      A(    ;
      O     I      0.2;
      O     M   1802.0;
      O     M    201.5;
      )     ;
      AN    M    201.7;
      A     M    201.6;
      A     M   1800.0;
      AN    M   1700.0;
      =     L      0.0;
      A     L      0.0;
      BLD   102;
      =     M    201.5;
      A     L      0.0;
      A     I      0.0;
      AN    I      0.1;
      =     M    201.4;
      A     L      0.0;
      AN    I      0.0;
      AN    I      0.1;
      =     M    202.0;
      A     L      0.0;
      AN    I      0.0;
      A     I      0.1;
      =     M    201.3;
NETWORK
TITLE =AUTO START

      A(    ;
      O     I      0.5;
      O     M   1802.1;
      O     M    201.2;
      )     ;
      A     M    201.4;
      A     I     68.1;
      A     I     69.0;
      AN    M    200.7;
      =     M    201.2;
NETWORK
TITLE =

      AN    M    201.7;
      AN    M    202.5;
      AN    M    601.1;
      AN    M    200.6;
      AN    M    820.0;
      NOT   ;
      =     M    200.7;
NETWORK
TITLE =AIR ERROR

      ON    I     31.2;
      O     ;
      A     M    201.7;
      AN    M    201.1;
      =     M    201.7;
NETWORK
TITLE =
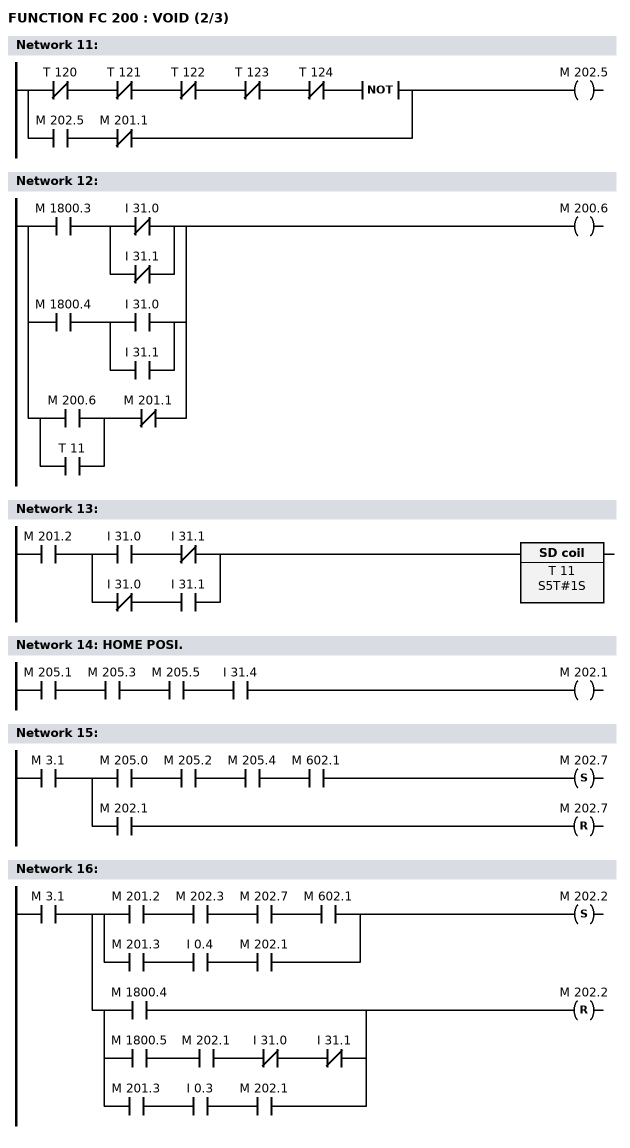

      AN    T    120;
      AN    T    121;
      AN    T    122;
      AN    T    123;
      AN    T    124;
      NOT   ;
      O     ;
      A     M    202.5;
      AN    M    201.1;
      =     M    202.5;
NETWORK
TITLE =

      A     M   1800.3;
      A(    ;
      ON    I     31.0;
      ON    I     31.1;
      )     ;
      O     ;
      A     M   1800.4;
      A(    ;
      O     I     31.0;
      O     I     31.1;
      )     ;
      O     ;
      A(    ;
      O     M    200.6;
      O     T     11;
      )     ;
      AN    M    201.1;
      =     M    200.6;
NETWORK
TITLE =

      A     M    201.2;
      A(    ;
      A     I     31.0;
      AN    I     31.1;
      O     ;
      AN    I     31.0;
      A     I     31.1;
      )     ;
      L     S5T#1S;
      SD    T     11;
NETWORK
TITLE =HOME POSI.

      A     M    205.1;
      A     M    205.3;
      A     M    205.5;
      A     I     31.4;
      =     M    202.1;
NETWORK
TITLE =

      A     M      3.1;
      =     L      0.0;
      A     L      0.0;
      A     M    205.0;
      A     M    205.2;
      A     M    205.4;
      A     M    602.1;
      S     M    202.7;
      A     L      0.0;
      A     M    202.1;
      R     M    202.7;
NETWORK
TITLE =

      A     M      3.1;
      =     L      0.0;
      A     L      0.0;
      A(    ;
      A     M    201.2;
      A     M    202.3;
      A     M    202.7;
      A     M    602.1;
      O     ;
      A     M    201.3;
      A     I      0.4;
      A     M    202.1;
      )     ;
      S     M    202.2;
      A     L      0.0;
      A(    ;
      O     M   1800.4;
      O     ;
      A     M   1800.5;
      A     M    202.1;
      AN    I     31.0;
      AN    I     31.1;
      O     ;
      A     M    201.3;
      A     I      0.3;
      A     M    202.1;
      )     ;
      R     M    202.2;
NETWORK
TITLE =
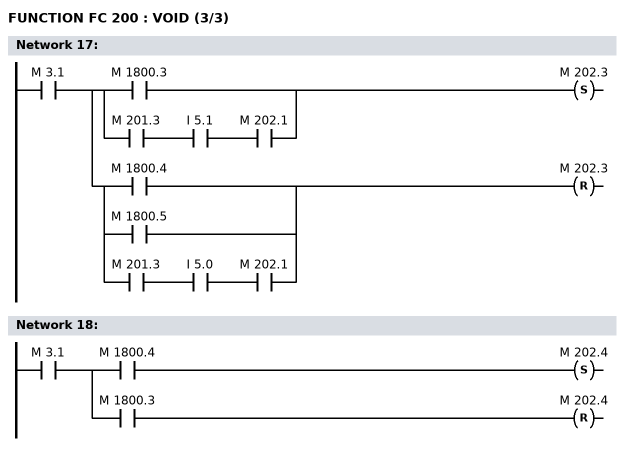

      A     M      3.1;
      =     L      0.0;
      A     L      0.0;
      A(    ;
      O     M   1800.3;
      O     ;
      A     M    201.3;
      A     I      5.1;
      A     M    202.1;
      )     ;
      S     M    202.3;
      A     L      0.0;
      A(    ;
      O     M   1800.4;
      O     M   1800.5;
      O     ;
      A     M    201.3;
      A     I      5.0;
      A     M    202.1;
      )     ;
      R     M    202.3;
NETWORK
TITLE =

      A     M      3.1;
      =     L      0.0;
      A     L      0.0;
      A     M   1800.4;
      S     M    202.4;
      A     L      0.0;
      A     M   1800.3;
      R     M    202.4;
NETWORK
TITLE =

      AN    OV;
      =     L      0.0;
      A     L      0.0;
      A(    ;
      O     M   1800.4;
      O     M   1801.0;
      )     ;
      S     M    207.0;
      A     L      0.0;
      A     T     70;
      R     M    207.0;
NETWORK
TITLE =CAM1 UP

      A     M    201.3;
      =     L      0.0;
      A     L      0.0;
      AN    I      3.5;
      =     L      0.1;
      A     L      0.1;
      AN    I      3.4;
      =     L      0.2;
      A     L      0.2;
      AN    I      3.3;
      A     I      3.2;
      =     M    203.0;
      A     L      0.2;
      A     I      3.3;
      AN    I      3.2;
      =     M    203.1;
      A     L      0.2;
      A     I      3.3;
      A     I      3.2;
      =     M    203.2;
      A     L      0.1;
      A     I      3.4;
      =     L      0.2;
      A     L      0.2;
      AN    I      3.3;
      =     L      0.3;
      A     L      0.3;
      AN    I      3.2;
      =     M    203.3;
      A     L      0.3;
      A     I      3.2;
      =     M    203.4;
      A     L      0.2;
      A     I      3.3;
      =     L      0.3;
      A     L      0.3;
      AN    I      3.2;
      =     M    203.5;
      A     L      0.3;
      A     I      3.2;
      =     M    203.6;
      A     L      0.0;
      A     I      3.4;
      AN    I      3.4;
      =     L      0.1;
      A     L      0.1;
      AN    I      3.3;
      =     L      0.2;
      A     L      0.2;
      AN    I      3.2;
      =     M    203.7;
      A     L      0.2;
      A     I      3.2;
      =     M    204.0;
      A     L      0.1;
      A     I      3.3;
      =     L      0.2;
      A     L      0.2;
      AN    I      3.2;
      =     M    204.1;
      A     L      0.2;
      A     I      3.2;
      =     M    204.2;
NETWORK
TITLE =핀/클램프 전_후진단
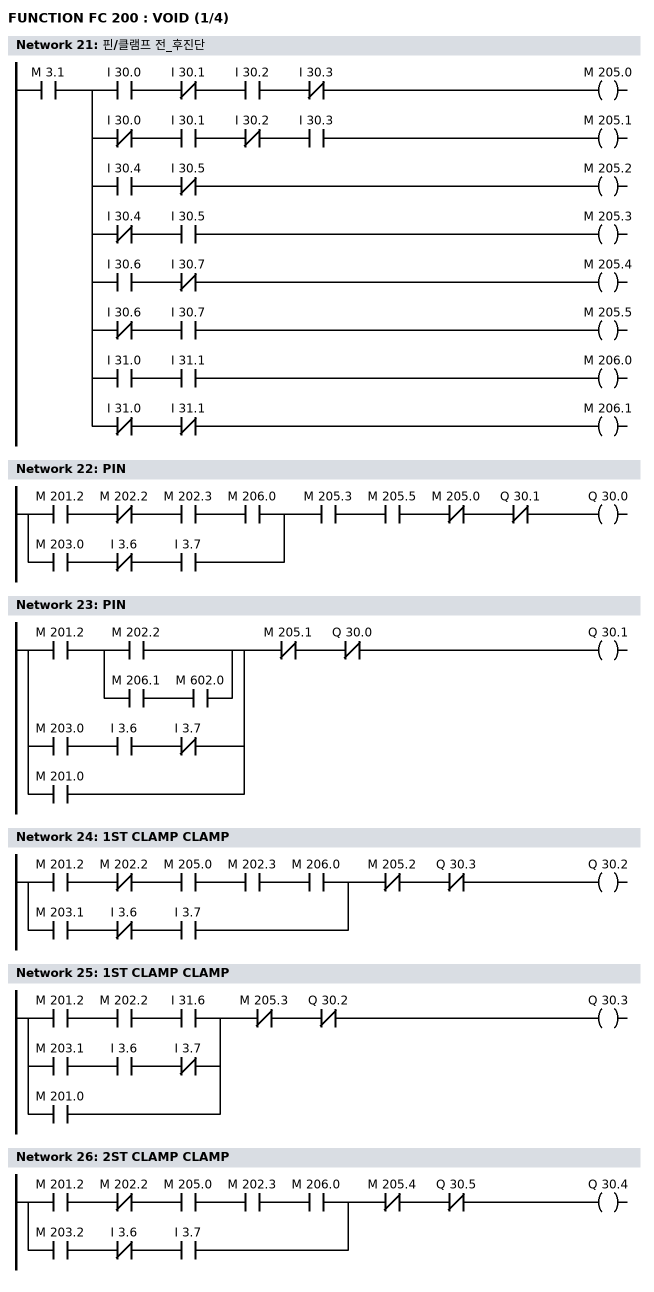

      A     M      3.1;
      =     L      0.0;
      A     L      0.0;
      A     I     30.0;
      AN    I     30.1;
      A     I     30.2;
      AN    I     30.3;
      =     M    205.0;
      A     L      0.0;
      AN    I     30.0;
      A     I     30.1;
      AN    I     30.2;
      A     I     30.3;
      =     M    205.1;
      A     L      0.0;
      A     I     30.4;
      AN    I     30.5;
      =     M    205.2;
      A     L      0.0;
      AN    I     30.4;
      A     I     30.5;
      =     M    205.3;
      A     L      0.0;
      A     I     30.6;
      AN    I     30.7;
      =     M    205.4;
      A     L      0.0;
      AN    I     30.6;
      A     I     30.7;
      =     M    205.5;
      A     L      0.0;
      A     I     31.0;
      A     I     31.1;
      =     M    206.0;
      A     L      0.0;
      AN    I     31.0;
      AN    I     31.1;
      =     M    206.1;
NETWORK
TITLE =PIN

      A(    ;
      A     M    201.2;
      AN    M    202.2;
      A     M    202.3;
      A     M    206.0;
      O     ;
      A     M    203.0;
      AN    I      3.6;
      A     I      3.7;
      )     ;
      A     M    205.3;
      A     M    205.5;
      AN    M    205.0;
      AN    Q     30.1;
      =     Q     30.0;
NETWORK
TITLE =PIN

      A(    ;
      A     M    201.2;
      A(    ;
      O     M    202.2;
      O     ;
      A     M    206.1;
      A     M    602.0;
      )     ;
      O     ;
      A     M    203.0;
      A     I      3.6;
      AN    I      3.7;
      O     M    201.0;
      )     ;
      AN    M    205.1;
      AN    Q     30.0;
      =     Q     30.1;
NETWORK
TITLE =1ST CLAMP CLAMP

      A(    ;
      A     M    201.2;
      AN    M    202.2;
      A     M    205.0;
      A     M    202.3;
      A     M    206.0;
      O     ;
      A     M    203.1;
      AN    I      3.6;
      A     I      3.7;
      )     ;
      AN    M    205.2;
      AN    Q     30.3;
      =     Q     30.2;
NETWORK
TITLE =1ST CLAMP CLAMP

      A(    ;
      A     M    201.2;
      A     M    202.2;
      A     I     31.6;
      O     ;
      A     M    203.1;
      A     I      3.6;
      AN    I      3.7;
      O     M    201.0;
      )     ;
      AN    M    205.3;
      AN    Q     30.2;
      =     Q     30.3;
NETWORK
TITLE =2ST CLAMP CLAMP

      A(    ;
      A     M    201.2;
      AN    M    202.2;
      A     M    205.0;
      A     M    202.3;
      A     M    206.0;
      O     ;
      A     M    203.2;
      AN    I      3.6;
      A     I      3.7;
      )     ;
      AN    M    205.4;
      AN    Q     30.5;
      =     Q     30.4;
NETWORK
TITLE =2ST CLAMP CLAMP
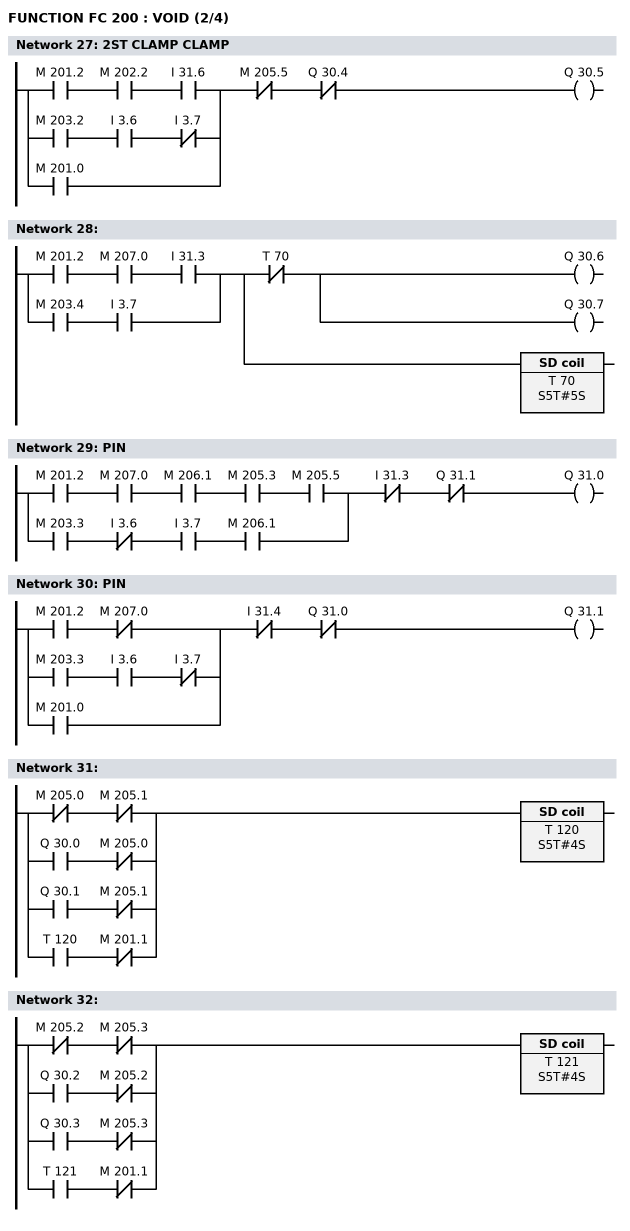

      A(    ;
      A     M    201.2;
      A     M    202.2;
      A     I     31.6;
      O     ;
      A     M    203.2;
      A     I      3.6;
      AN    I      3.7;
      O     M    201.0;
      )     ;
      AN    M    205.5;
      AN    Q     30.4;
      =     Q     30.5;
NETWORK
TITLE =

      A     M    201.2;
      A     M    207.0;
      A     I     31.3;
      O     ;
      A     M    203.4;
      A     I      3.7;
      =     L      0.0;
      A     L      0.0;
      AN    T     70;
      =     Q     30.6;
      =     Q     30.7;
      A     L      0.0;
      BLD   102;
      L     S5T#5S;
      SD    T     70;
NETWORK
TITLE =PIN

      A(    ;
      A     M    201.2;
      A     M    207.0;
      A     M    206.1;
      A     M    205.3;
      A     M    205.5;
      O     ;
      A     M    203.3;
      AN    I      3.6;
      A     I      3.7;
      A     M    206.1;
      )     ;
      AN    I     31.3;
      AN    Q     31.1;
      =     Q     31.0;
NETWORK
TITLE =PIN

      A(    ;
      A     M    201.2;
      AN    M    207.0;
      O     ;
      A     M    203.3;
      A     I      3.6;
      AN    I      3.7;
      O     M    201.0;
      )     ;
      AN    I     31.4;
      AN    Q     31.0;
      =     Q     31.1;
NETWORK
TITLE =

      AN    M    205.0;
      AN    M    205.1;
      O     ;
      A     Q     30.0;
      AN    M    205.0;
      O     ;
      A     Q     30.1;
      AN    M    205.1;
      O     ;
      A     T    120;
      AN    M    201.1;
      L     S5T#4S;
      SD    T    120;
NETWORK
TITLE =

      AN    M    205.2;
      AN    M    205.3;
      O     ;
      A     Q     30.2;
      AN    M    205.2;
      O     ;
      A     Q     30.3;
      AN    M    205.3;
      O     ;
      A     T    121;
      AN    M    201.1;
      L     S5T#4S;
      SD    T    121;
NETWORK
TITLE =
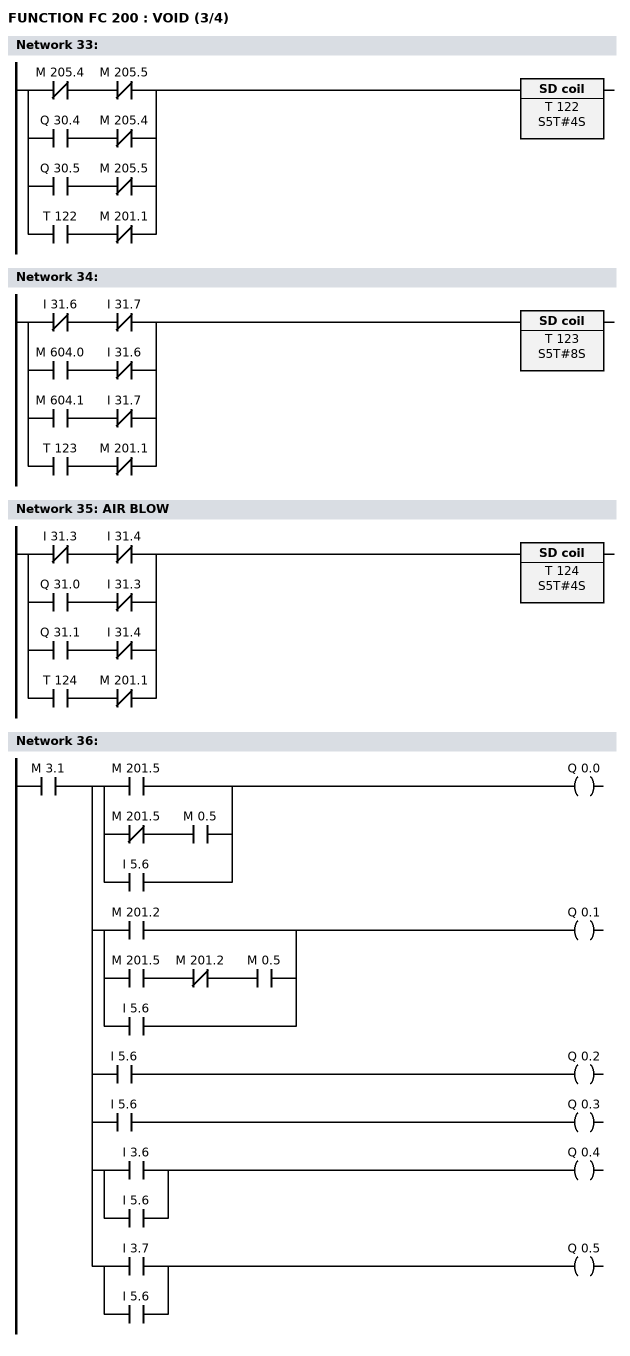

      AN    M    205.4;
      AN    M    205.5;
      O     ;
      A     Q     30.4;
      AN    M    205.4;
      O     ;
      A     Q     30.5;
      AN    M    205.5;
      O     ;
      A     T    122;
      AN    M    201.1;
      L     S5T#4S;
      SD    T    122;
NETWORK
TITLE =

      AN    I     31.6;
      AN    I     31.7;
      O     ;
      A     M    604.0;
      AN    I     31.6;
      O     ;
      A     M    604.1;
      AN    I     31.7;
      O     ;
      A     T    123;
      AN    M    201.1;
      L     S5T#8S;
      SD    T    123;
NETWORK
TITLE =AIR BLOW

      AN    I     31.3;
      AN    I     31.4;
      O     ;
      A     Q     31.0;
      AN    I     31.3;
      O     ;
      A     Q     31.1;
      AN    I     31.4;
      O     ;
      A     T    124;
      AN    M    201.1;
      L     S5T#4S;
      SD    T    124;
NETWORK
TITLE =

      A     M      3.1;
      =     L      0.0;
      A     L      0.0;
      A(    ;
      O     M    201.5;
      O     ;
      AN    M    201.5;
      A     M      0.5;
      O     I      5.6;
      )     ;
      =     Q      0.0;
      A     L      0.0;
      A(    ;
      O     M    201.2;
      O     ;
      A     M    201.5;
      AN    M    201.2;
      A     M      0.5;
      O     I      5.6;
      )     ;
      =     Q      0.1;
      A     L      0.0;
      A     I      5.6;
      =     Q      0.2;
      A     L      0.0;
      A     I      5.6;
      =     Q      0.3;
      A     L      0.0;
      A(    ;
      O     I      3.6;
      O     I      5.6;
      )     ;
      =     Q      0.4;
      A     L      0.0;
      A(    ;
      O     I      3.7;
      O     I      5.6;
      )     ;
      =     Q      0.5;
NETWORK
TITLE =메인제어반1 에어이상 램프
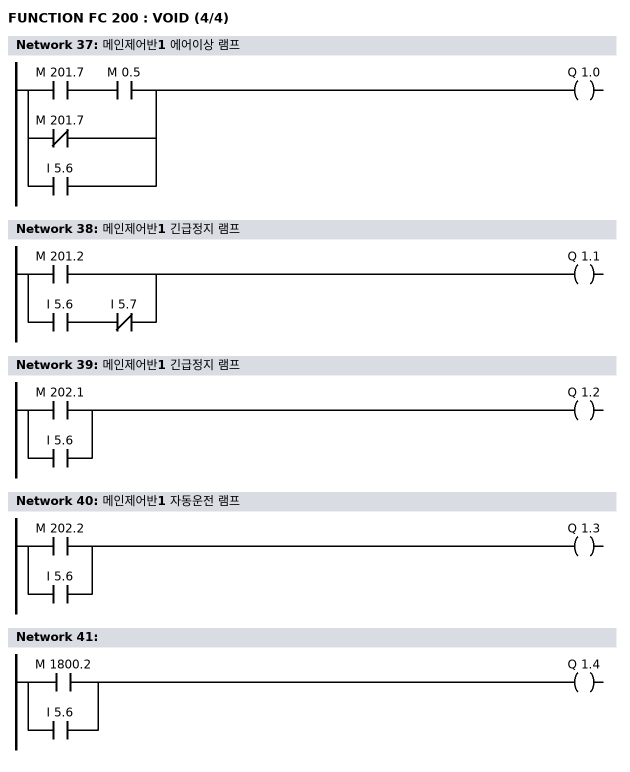

      A     M    201.7;
      A     M      0.5;
      ON    M    201.7;
      O     I      5.6;
      =     Q      1.0;
NETWORK
TITLE =메인제어반1 긴급정지 램프

      O     M    201.2;
      O     ;
      A     I      5.6;
      AN    I      5.7;
      =     Q      1.1;
NETWORK
TITLE =메인제어반1 긴급정지 램프

      O     M    202.1;
      O     I      5.6;
      =     Q      1.2;
NETWORK
TITLE =메인제어반1 자동운전 램프

      O     M    202.2;
      O     I      5.6;
      =     Q      1.3;
NETWORK
TITLE =

      O     M   1800.2;
      O     I      5.6;
      =     Q      1.4;
NETWORK
TITLE =

      A     DB486.DBX   21.1;
      A     OV;
      O     I      5.6;
      =     Q      1.5;
NETWORK
TITLE =
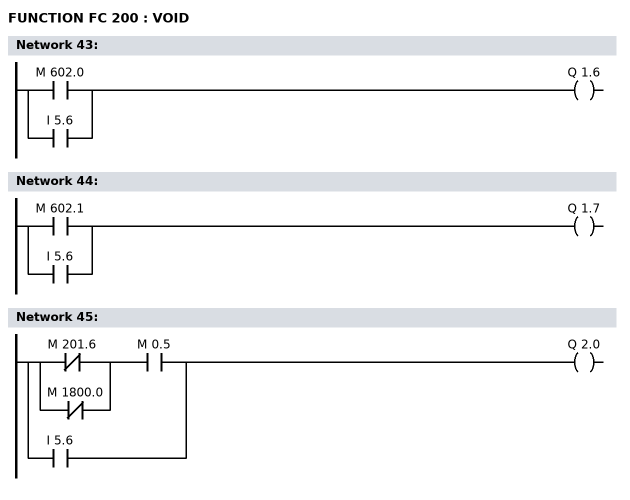

      O     M    602.0;
      O     I      5.6;
      =     Q      1.6;
NETWORK
TITLE =

      O     M    602.1;
      O     I      5.6;
      =     Q      1.7;
NETWORK
TITLE =

      A(    ;
      ON    M    201.6;
      ON    M   1800.0;
      )     ;
      A     M      0.5;
      O     I      5.6;
      =     Q      2.0;
NETWORK
TITLE =

      A     M    202.5;
      A     OV;
      O     I      5.6;
      =     Q      2.1;
NETWORK
TITLE =
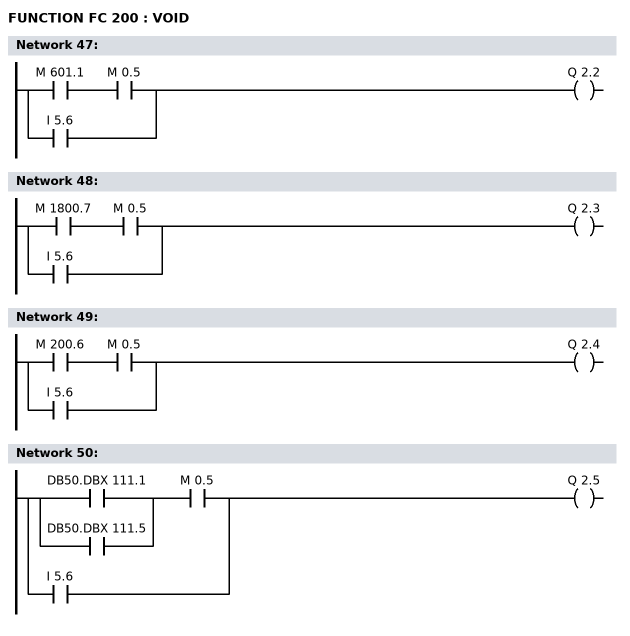

      A     M    601.1;
      A     M      0.5;
      O     I      5.6;
      =     Q      2.2;
NETWORK
TITLE =

      A     M   1800.7;
      A     M      0.5;
      O     I      5.6;
      =     Q      2.3;
NETWORK
TITLE =

      A     M    200.6;
      A     M      0.5;
      O     I      5.6;
      =     Q      2.4;
NETWORK
TITLE =

      A(    ;
      O     DB50.DBX  111.1;
      O     DB50.DBX  111.5;
      )     ;
      A     M      0.5;
      O     I      5.6;
      =     Q      2.5;
NETWORK
TITLE =

      A     OV;
      A     M      0.5;
      O     I      5.6;
      =     Q      2.6;
NETWORK
TITLE =

      A     OV;
      A     M      0.5;
      O     I      5.6;
      =     Q      2.7;
NETWORK
TITLE =부저울림
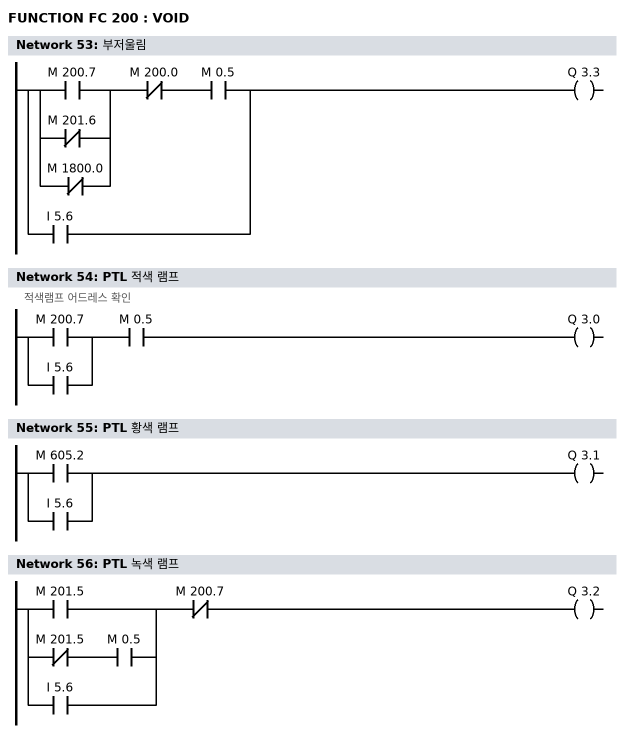

      A(    ;
      O     M    200.7;
      ON    M    201.6;
      ON    M   1800.0;
      )     ;
      AN    M    200.0;
      A     M      0.5;
      O     I      5.6;
      =     Q      3.3;
NETWORK
TITLE =PTL 적색 램프
//적색램프 어드레스 확인
      A(    ;
      O     M    200.7;
      O     I      5.6;
      )     ;
      A     M      0.5;
      =     Q      3.0;
NETWORK
TITLE =PTL 황색 램프

      O     M    605.2;
      O     I      5.6;
      =     Q      3.1;
NETWORK
TITLE =PTL 녹색 램프

      A(    ;
      O     M    201.5;
      O     ;
      AN    M    201.5;
      A     M      0.5;
      O     I      5.6;
      )     ;
      AN    M    200.7;
      =     Q      3.2;
END_FUNCTION

FUNCTION FC 210 : VOID
TITLE =
VERSION : 0.1

BEGIN
NETWORK
TITLE =#708-1 STN

      AN    OV;
      =     L      0.0;
      A     L      0.0;
      JNB   _001;
      L     IW    30;
      T     DB50.DBW   30;
_001: NOP   0;
      A     L      0.0;
      JNB   _002;
      L     QW    30;
      T     DB50.DBW   40;
_002: NOP   0;
NETWORK
TITLE =공정 인터록

      AN    OV;
      =     L      0.0;
      A     L      0.0;
      JNB   _003;
      L     MD  1800;
      T     DB50.DBD  120;
_003: NOP   0;
      A     L      0.0;
      JNB   _004;
      L     MD  1900;
      T     DB50.DBD  124;
_004: NOP   0;
NETWORK
TITLE =

      AN    OV;
      =     L      0.0;
      A     L      0.0;
      AN    T      5;
      L     S5T#1S;
      SD    T      6;
      A     L      0.0;
      A     T      6;
      L     S5T#1S;
      SD    T      5;
NETWORK
TITLE =

      AN    OV;
      =     L      0.0;
      A     L      0.0;
      A(    ;
      A     M    205.0;
      AN    T    120;
      O     ;
      A     T    120;
      A     T      6;
      )     ;
      =     DB50.DBX   60.0;
      A     L      0.0;
      A(    ;
      A     M    205.1;
      AN    T    120;
      O     ;
      A     T    120;
      A     T      6;
      )     ;
      =     DB50.DBX   60.1;
      A     L      0.0;
      A(    ;
      A     M    205.2;
      AN    T    121;
      O     ;
      A     T    121;
      A     T      6;
      )     ;
      =     DB50.DBX   60.2;
      A     L      0.0;
      A(    ;
      A     M    205.3;
      AN    T    121;
      O     ;
      A     T    121;
      A     T      6;
      )     ;
      =     DB50.DBX   60.3;
      A     L      0.0;
      A(    ;
      A     M    205.4;
      AN    T    122;
      O     ;
      A     T    122;
      A     T      6;
      )     ;
      =     DB50.DBX   60.4;
      A     L      0.0;
      A(    ;
      A     M    205.5;
      AN    T    122;
      O     ;
      A     T    122;
      A     T      6;
      )     ;
      =     DB50.DBX   60.5;
      A     L      0.0;
      A(    ;
      A     I     31.6;
      AN    T    123;
      O     ;
      A     T    123;
      A     T      6;
      )     ;
      =     DB50.DBX   60.6;
      A     L      0.0;
      A(    ;
      A     I     31.7;
      AN    T    123;
      O     ;
      A     T    123;
      A     T      6;
      )     ;
      =     DB50.DBX   60.7;
NETWORK
TITLE =

      AN    OV;
      =     L      0.0;
      A     L      0.0;
      A(    ;
      A     I     31.3;
      AN    T    124;
      O     ;
      A     T    124;
      A     T      6;
      )     ;
      =     DB50.DBX   61.0;
      A     L      0.0;
      A(    ;
      A     I     31.4;
      AN    T    124;
      O     ;
      A     T    124;
      A     T      6;
      )     ;
      =     DB50.DBX   61.1;
      A     L      0.0;
      A     OV;
      =     DB50.DBX   61.2;
      A     L      0.0;
      A     OV;
      =     DB50.DBX   61.3;
      A     L      0.0;
      A(    ;
      O     DB50.DBX  111.1;
      O     DB50.DBX  111.5;
      )     ;
      A     T      6;
      =     DB50.DBX   61.4;
      A     L      0.0;
      A     OV;
      =     DB50.DBX   61.5;
      A     L      0.0;
      A     M    206.0;
      =     DB50.DBX   61.6;
      A     L      0.0;
      AN    M    206.0;
      =     DB50.DBX   61.7;
NETWORK
TITLE =

      AN    OV;
      =     L      0.0;
      A     L      0.0;
      A     M    202.2;
      =     DB50.DBX   62.2;
      A     L      0.0;
      A     M    202.1;
      =     DB50.DBX   62.3;
      A     L      0.0;
      A     M   1900.2;
      =     DB50.DBX   62.4;
      A     L      0.0;
      A     M   1800.2;
      =     DB50.DBX   62.5;
      A     L      0.0;
      A     M   1900.3;
      =     DB50.DBX   62.6;
      A     L      0.0;
      A     M    202.3;
      =     DB50.DBX   62.7;
NETWORK
TITLE =

      AN    OV;
      =     L      0.0;
      A     L      0.0;
      A     M   1900.4;
      =     DB50.DBX   63.0;
      A     L      0.0;
      A     M    202.4;
      =     DB50.DBX   63.1;
      A     L      0.0;
      A     OV;
      =     DB50.DBX   63.2;
      A     L      0.0;
      A     OV;
      =     DB50.DBX   63.3;
      A     L      0.0;
      A     OV;
      =     DB50.DBX   63.4;
      A     L      0.0;
      A     OV;
      =     DB50.DBX   63.5;
NETWORK
TITLE =

      AN    OV;
      =     L      0.0;
      A     L      0.0;
      A     I     69.0;
      =     DB50.DBX   64.0;
      A     L      0.0;
      A     I     69.1;
      =     DB50.DBX   64.1;
      A     L      0.0;
      A     I     69.2;
      =     DB50.DBX   64.2;
      A     L      0.0;
      A     I     69.3;
      =     DB50.DBX   64.3;
NETWORK
TITLE =L/S 이상

      AN    OV;
      =     L      0.0;
      A     L      0.0;
      A     T    120;
      A     T      6;
      =     DB50.DBX   65.0;
      A     L      0.0;
      A     T    121;
      A     T      6;
      =     DB50.DBX   65.1;
      A     L      0.0;
      A     T    122;
      A     T      6;
      =     DB50.DBX   65.2;
      A     L      0.0;
      A     T    123;
      A     T      6;
      =     DB50.DBX   65.3;
      A     L      0.0;
      A     T    124;
      A     T      6;
      =     DB50.DBX   65.4;
      A     L      0.0;
      A     M    200.6;
      A     T      6;
      =     DB50.DBX   65.5;
      A     L      0.0;
      A     OV;
      =     DB50.DBX   65.6;
      A     L      0.0;
      A     OV;
      =     DB50.DBX   65.7;
NETWORK
TITLE =GP  DP이상표시(1-8)
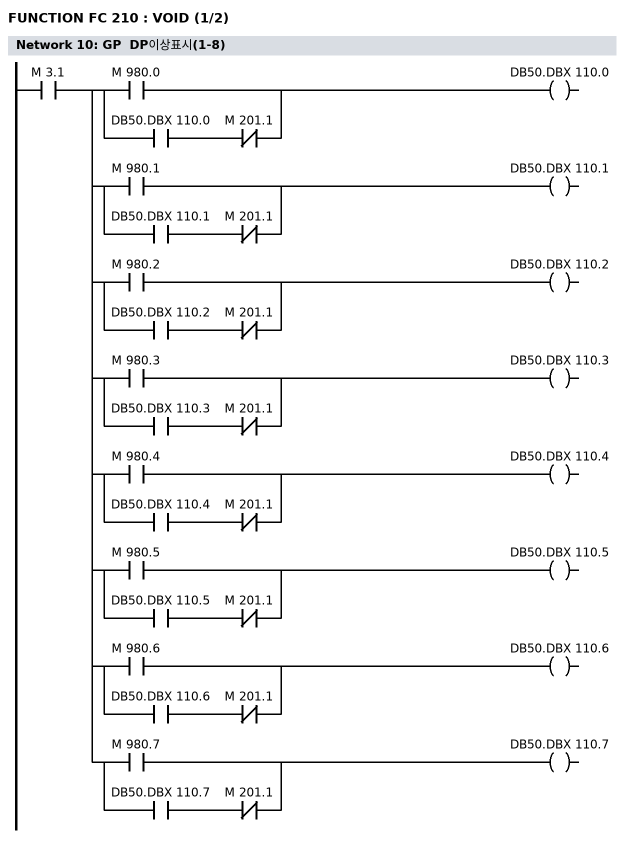

      A     M      3.1;
      =     L      0.0;
      A     L      0.0;
      A(    ;
      O     M    980.0;
      O     ;
      A     DB50.DBX  110.0;
      AN    M    201.1;
      )     ;
      =     DB50.DBX  110.0;
      A     L      0.0;
      A(    ;
      O     M    980.1;
      O     ;
      A     DB50.DBX  110.1;
      AN    M    201.1;
      )     ;
      =     DB50.DBX  110.1;
      A     L      0.0;
      A(    ;
      O     M    980.2;
      O     ;
      A     DB50.DBX  110.2;
      AN    M    201.1;
      )     ;
      =     DB50.DBX  110.2;
      A     L      0.0;
      A(    ;
      O     M    980.3;
      O     ;
      A     DB50.DBX  110.3;
      AN    M    201.1;
      )     ;
      =     DB50.DBX  110.3;
      A     L      0.0;
      A(    ;
      O     M    980.4;
      O     ;
      A     DB50.DBX  110.4;
      AN    M    201.1;
      )     ;
      =     DB50.DBX  110.4;
      A     L      0.0;
      A(    ;
      O     M    980.5;
      O     ;
      A     DB50.DBX  110.5;
      AN    M    201.1;
      )     ;
      =     DB50.DBX  110.5;
      A     L      0.0;
      A(    ;
      O     M    980.6;
      O     ;
      A     DB50.DBX  110.6;
      AN    M    201.1;
      )     ;
      =     DB50.DBX  110.6;
      A     L      0.0;
      A(    ;
      O     M    980.7;
      O     ;
      A     DB50.DBX  110.7;
      AN    M    201.1;
      )     ;
      =     DB50.DBX  110.7;
NETWORK
TITLE =GP  DP이상표시(9-16)
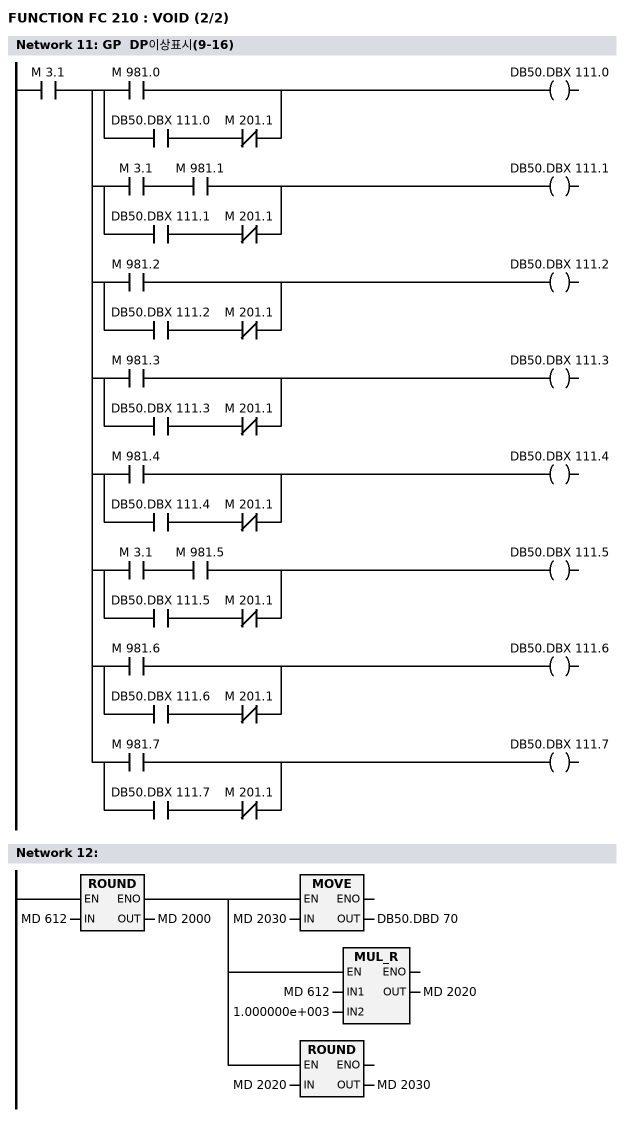

      A     M      3.1;
      =     L      0.0;
      A     L      0.0;
      A(    ;
      O     M    981.0;
      O     ;
      A     DB50.DBX  111.0;
      AN    M    201.1;
      )     ;
      =     DB50.DBX  111.0;
      A     L      0.0;
      A(    ;
      A     M      3.1;
      A     M    981.1;
      O     ;
      A     DB50.DBX  111.1;
      AN    M    201.1;
      )     ;
      =     DB50.DBX  111.1;
      A     L      0.0;
      A(    ;
      O     M    981.2;
      O     ;
      A     DB50.DBX  111.2;
      AN    M    201.1;
      )     ;
      =     DB50.DBX  111.2;
      A     L      0.0;
      A(    ;
      O     M    981.3;
      O     ;
      A     DB50.DBX  111.3;
      AN    M    201.1;
      )     ;
      =     DB50.DBX  111.3;
      A     L      0.0;
      A(    ;
      O     M    981.4;
      O     ;
      A     DB50.DBX  111.4;
      AN    M    201.1;
      )     ;
      =     DB50.DBX  111.4;
      A     L      0.0;
      A(    ;
      A     M      3.1;
      A     M    981.5;
      O     ;
      A     DB50.DBX  111.5;
      AN    M    201.1;
      )     ;
      =     DB50.DBX  111.5;
      A     L      0.0;
      A(    ;
      O     M    981.6;
      O     ;
      A     DB50.DBX  111.6;
      AN    M    201.1;
      )     ;
      =     DB50.DBX  111.6;
      A     L      0.0;
      A(    ;
      O     M    981.7;
      O     ;
      A     DB50.DBX  111.7;
      AN    M    201.1;
      )     ;
      =     DB50.DBX  111.7;
NETWORK
TITLE =

      L     MD   612;
      RND   ;
      T     MD  2000;
      AN    OV;
      SAVE  ;
      CLR   ;
      A     BR;
      =     L      0.0;
      A     L      0.0;
      JNB   _005;
      L     MD  2030;
      T     DB50.DBD   70;
_005: NOP   0;
      A     L      0.0;
      JNB   _006;
      L     MD   612;
      L     1.000000e+003;
      *R    ;
      T     MD  2020;
_006: NOP   0;
      A     L      0.0;
      JNB   _007;
      L     MD  2020;
      RND   ;
      T     MD  2030;
_007: NOP   0;
END_FUNCTION

FUNCTION FC 324 : VOID
TITLE =
VERSION : 0.1

BEGIN
NETWORK
TITLE =DP DIAGNOSTIC FOR DP MASTER SYSTEM(1)

      AN    OV;
      =     L      0.0;
      BLD   103;
      A     OV;
      =     L      0.1;
      BLD   103;
      CALL FC   325 (
           CHECK_ACTIV              := L      0.0,
           EXTERNAL_DP_INTERFACE    := L      0.1,
           DP_MASTERSYSTEM          := 1,
           DATA_FIELD               := P#DB325.DBX0.0 BYTE 50,
           SUM_SLAVES_DIAG          := DB325.DBW   82,
           LIST_SLAVES_NOT_PRESENT  := P#DB325.DBX 50.0 DWORD 4,
           LIST_SLAVES_ERROR        := P#DB325.DBX 66.0 DWORD 4,
           RETVAL                   := DB325.DBW   84,
           BUSY                     := DB325.DBX   90.0);
      NOP   0;
NETWORK
TITLE =

      O     DB325.DBX   51.1;
      O     DB325.DBX   67.1;
      O     ;
      A     M    801.1;
      A(    ;
      ON    M    201.1;
      ON    OV;
      )     ;
      =     M    801.1;
NETWORK
TITLE =

      O     DB325.DBX   51.5;
      O     DB325.DBX   67.5;
      O     ;
      A     M    801.5;
      A(    ;
      ON    M    201.1;
      ON    OV;
      )     ;
      =     M    801.5;
NETWORK
TITLE =

      AN    M    801.1;
      AN    M    801.5;
      NOT   ;
      A     OV;
      =     M    820.0;
END_FUNCTION

DATA_BLOCK DB 71
TITLE =
AUTHOR : SIMATIC
FAMILY : CP300PBK
VERSION : 0.0

 FB 12
BEGIN
   REQ := FALSE;
   R := FALSE;
   ID := W#16#0;
   R_ID := DW#16#0;
   DONE := FALSE;
   ERROR := FALSE;
   STATUS := W#16#0;
   LEN := W#16#0;
   FB_ZUSTAND := B#16#0;
   REQ_SAVE := FALSE;
   R_SAVE := FALSE;
   ID_SAVE := W#16#0;
   R_ID_SAVE := DW#16#0;
   LEN_SAVE := W#16#0;
   SD_1_SAVE0 := W#16#0;
   SD_1_SAVE2 := W#16#0;
   SD_1_SAVE4 := W#16#0;
   SD_1_SAVE6 := W#16#0;
   SD_1_SAVE8 := W#16#0;
   HS_REQ_BYTE.rii := FALSE;
   HS_REQ_BYTE.nva := FALSE;
   HS_REQ_BYTE.ofs := FALSE;
   HS_REQ_BYTE.dir := FALSE;
   HS_REQ_BYTE.res := FALSE;
   HS_REQ_BYTE.roc := FALSE;
   HS_REQ_BYTE.nls := FALSE;
   HS_REQ_BYTE.rlo := FALSE;
   HS_RESP_BYTE.aii := FALSE;
   HS_RESP_BYTE.sns := FALSE;
   HS_RESP_BYTE.sqc := FALSE;
   HS_RESP_BYTE.ads := FALSE;
   HS_RESP_BYTE.aoc := FALSE;
   HS_RESP_BYTE.rs1 := FALSE;
   HS_RESP_BYTE.cnr := FALSE;
   HS_RESP_BYTE.rs2 := FALSE;
   HS_RESP_DSNR := B#16#0;
   HS_RESP_OFFSET := W#16#0;
   SD_1_WORD0 := W#16#0;
   SD_1_COUNT := W#16#0;
   SD_1_DBNUMMER := W#16#0;
   SD_1_DWORD6 := DW#16#0;
   SD_1_TYP := B#16#0;
   SFC_PARAM.LEN := W#16#0;
   SFC_PARAM.DB_NUMMER := W#16#0;
   SFC_PARAM.START := DW#16#0;
   BUFFER[0] := W#16#0;
   BUFFER[1] := W#16#0;
   BUFFER[2] := W#16#0;
   BUFFER[3] := W#16#0;
   BUFFER[4] := W#16#0;
   BUFFER[5] := W#16#0;
   BUFFER[6] := W#16#0;
   BUFFER[7] := W#16#0;
   BUFFER[8] := W#16#0;
   BUFFER[9] := W#16#0;
   BUFFER[10] := W#16#0;
   BUFFER[11] := W#16#0;
   BUFFER[12] := W#16#0;
   BUFFER[13] := W#16#0;
   BUFFER[14] := W#16#0;
   BUFFER[15] := W#16#0;
   BUFFER[16] := W#16#0;
   BUFFER[17] := W#16#0;
   BUFFER[18] := W#16#0;
   BUFFER[19] := W#16#0;
   BUFFER[20] := W#16#0;
   BUFFER[21] := W#16#0;
   BUFFER[22] := W#16#0;
   BUFFER[23] := W#16#0;
   BUFFER[24] := W#16#0;
   BUFFER[25] := W#16#0;
   BUFFER[26] := W#16#0;
   BUFFER[27] := W#16#0;
   BUFFER[28] := W#16#0;
   BUFFER[29] := W#16#0;
   BUFFER[30] := W#16#0;
   BUFFER[31] := W#16#0;
   BUFFER[32] := W#16#0;
   BUFFER[33] := W#16#0;
   BUFFER[34] := W#16#0;
   BUFFER[35] := W#16#0;
   BUFFER[36] := W#16#0;
   BUFFER[37] := W#16#0;
   BUFFER[38] := W#16#0;
   BUFFER[39] := W#16#0;
   BUFFER[40] := W#16#0;
   BUFFER[41] := W#16#0;
   BUFFER[42] := W#16#0;
   BUFFER[43] := W#16#0;
   BUFFER[44] := W#16#0;
   BUFFER[45] := W#16#0;
   BUFFER[46] := W#16#0;
   BUFFER[47] := W#16#0;
   BUFFER[48] := W#16#0;
   BUFFER[49] := W#16#0;
   BUFFER[50] := W#16#0;
   BUFFER[51] := W#16#0;
   BUFFER[52] := W#16#0;
   BUFFER[53] := W#16#0;
   BUFFER[54] := W#16#0;
   BUFFER[55] := W#16#0;
   BUFFER[56] := W#16#0;
   BUFFER[57] := W#16#0;
   BUFFER[58] := W#16#0;
   BUFFER[59] := W#16#0;
   BUFFER[60] := W#16#0;
   BUFFER[61] := W#16#0;
   BUFFER[62] := W#16#0;
   BUFFER[63] := W#16#0;
   BUFFER[64] := W#16#0;
   BUFFER[65] := W#16#0;
   BUFFER[66] := W#16#0;
   BUFFER[67] := W#16#0;
   BUFFER[68] := W#16#0;
   BUFFER[69] := W#16#0;
   BUFFER[70] := W#16#0;
   BUFFER[71] := W#16#0;
   BUFFER[72] := W#16#0;
   BUFFER[73] := W#16#0;
   BUFFER[74] := W#16#0;
   BUFFER[75] := W#16#0;
   BUFFER[76] := W#16#0;
   BUFFER[77] := W#16#0;
   BUFFER[78] := W#16#0;
   BUFFER[79] := W#16#0;
   BUFFER[80] := W#16#0;
   BUFFER[81] := W#16#0;
   BUFFER[82] := W#16#0;
   BUFFER[83] := W#16#0;
   BUFFER[84] := W#16#0;
   BUFFER[85] := W#16#0;
   BUFFER[86] := W#16#0;
   BUFFER[87] := W#16#0;
   BUFFER[88] := W#16#0;
   BUFFER[89] := W#16#0;
   BUFFER[90] := W#16#0;
   BUFFER[91] := W#16#0;
   BUFFER[92] := W#16#0;
   BUFFER[93] := W#16#0;
   BUFFER[94] := W#16#0;
   BUFFER[95] := W#16#0;
   BUFFER[96] := W#16#0;
   BUFFER[97] := W#16#0;
   BUFFER[98] := W#16#0;
   BUFFER[99] := W#16#0;
   BUFFER[100] := W#16#0;
   BUFFER[101] := W#16#0;
   BUFFER[102] := W#16#0;
   BUFFER[103] := W#16#0;
   BUFFER[104] := W#16#0;
   BUFFER[105] := W#16#0;
   BUFFER[106] := W#16#0;
   BUFFER[107] := W#16#0;
   BUFFER[108] := W#16#0;
   BUFFER[109] := W#16#0;
   BUFFER[110] := W#16#0;
   BUFFER[111] := W#16#0;
   BUFFER[112] := W#16#0;
   BUFFER[113] := W#16#0;
   BUFFER[114] := W#16#0;
   BUFFER[115] := W#16#0;
   BUFFER[116] := W#16#0;
   BUFFER[117] := W#16#0;
   BUFFER[118] := W#16#0;
   BUFFER[119] := W#16#0;
   REASON_FOR_CLOSE := B#16#0;
   DS_NR := B#16#0;
   PARAM_OFFSET := B#16#0;
   MAX_PUFF_LEN_SAVE := W#16#0;
   TYP_BOOL := FALSE;
   KANAL_PROBLEM := FALSE;
   KOMM_PROBLEM := FALSE;
   SEND_STARTED := FALSE;
   RECV_STARTED := FALSE;
   RESET_REQUEST := FALSE;
   RESET_EXECUTED := FALSE;
   DS200_BUSY := FALSE;
   MAX_DATA_LEN := W#16#0;
   LADDR_PTR := DW#16#0;
   FC_DATA_LEN := W#16#0;
   LADDR := W#16#0;
   SLEEP := B#16#0;
   SLEEP_EXT := B#16#0;
   ID_CLOSE := W#16#0;
   FB_KENNUNG := B#16#F1;
END_DATA_BLOCK

DATA_BLOCK DB 81
TITLE =
AUTHOR : SIMATIC
FAMILY : CP300PBK
VERSION : 0.0

 FB 13
BEGIN
   EN_R := FALSE;
   ID := W#16#0;
   R_ID := DW#16#0;
   NDR := FALSE;
   ERROR := FALSE;
   STATUS := W#16#0;
   LEN := W#16#0;
   FB_ZUSTAND := B#16#0;
   EN_R_SAVE := FALSE;
   ID_SAVE := W#16#0;
   R_ID_SAVE := DW#16#0;
   FC_DATA_LEN := W#16#0;
   SD_1_SAVE0 := W#16#0;
   SD_1_SAVE2 := W#16#0;
   SD_1_SAVE4 := W#16#0;
   SD_1_SAVE6 := W#16#0;
   SD_1_SAVE8 := W#16#0;
   HS_REQ_BYTE.rii := FALSE;
   HS_REQ_BYTE.nva := FALSE;
   HS_REQ_BYTE.ofs := FALSE;
   HS_REQ_BYTE.dir := FALSE;
   HS_REQ_BYTE.res := FALSE;
   HS_REQ_BYTE.roc := FALSE;
   HS_REQ_BYTE.nls := FALSE;
   HS_REQ_BYTE.rlo := FALSE;
   HS_RESP_BYTE.aii := FALSE;
   HS_RESP_BYTE.sns := FALSE;
   HS_RESP_BYTE.sqc := FALSE;
   HS_RESP_BYTE.ads := FALSE;
   HS_RESP_BYTE.aoc := FALSE;
   HS_RESP_BYTE.rs1 := FALSE;
   HS_RESP_BYTE.cnr := FALSE;
   HS_RESP_BYTE.rs2 := FALSE;
   HS_RESP_DSNR := B#16#0;
   HS_RESP_OFFSET := W#16#0;
   SD_1_WORD0 := W#16#0;
   SD_1_COUNT := W#16#0;
   SD_1_DBNUMMER := W#16#0;
   SD_1_DWORD6 := DW#16#0;
   SD_1_TYP := B#16#0;
   SFC_PARAM.LEN := W#16#0;
   SFC_PARAM.DB_NUMMER := W#16#0;
   SFC_PARAM.START := DW#16#0;
   BUFFER[0] := W#16#0;
   BUFFER[1] := W#16#0;
   BUFFER[2] := W#16#0;
   BUFFER[3] := W#16#0;
   BUFFER[4] := W#16#0;
   BUFFER[5] := W#16#0;
   BUFFER[6] := W#16#0;
   BUFFER[7] := W#16#0;
   BUFFER[8] := W#16#0;
   BUFFER[9] := W#16#0;
   BUFFER[10] := W#16#0;
   BUFFER[11] := W#16#0;
   BUFFER[12] := W#16#0;
   BUFFER[13] := W#16#0;
   BUFFER[14] := W#16#0;
   BUFFER[15] := W#16#0;
   BUFFER[16] := W#16#0;
   BUFFER[17] := W#16#0;
   BUFFER[18] := W#16#0;
   BUFFER[19] := W#16#0;
   BUFFER[20] := W#16#0;
   BUFFER[21] := W#16#0;
   BUFFER[22] := W#16#0;
   BUFFER[23] := W#16#0;
   BUFFER[24] := W#16#0;
   BUFFER[25] := W#16#0;
   BUFFER[26] := W#16#0;
   BUFFER[27] := W#16#0;
   BUFFER[28] := W#16#0;
   BUFFER[29] := W#16#0;
   BUFFER[30] := W#16#0;
   BUFFER[31] := W#16#0;
   BUFFER[32] := W#16#0;
   BUFFER[33] := W#16#0;
   BUFFER[34] := W#16#0;
   BUFFER[35] := W#16#0;
   BUFFER[36] := W#16#0;
   BUFFER[37] := W#16#0;
   BUFFER[38] := W#16#0;
   BUFFER[39] := W#16#0;
   BUFFER[40] := W#16#0;
   BUFFER[41] := W#16#0;
   BUFFER[42] := W#16#0;
   BUFFER[43] := W#16#0;
   BUFFER[44] := W#16#0;
   BUFFER[45] := W#16#0;
   BUFFER[46] := W#16#0;
   BUFFER[47] := W#16#0;
   BUFFER[48] := W#16#0;
   BUFFER[49] := W#16#0;
   BUFFER[50] := W#16#0;
   BUFFER[51] := W#16#0;
   BUFFER[52] := W#16#0;
   BUFFER[53] := W#16#0;
   BUFFER[54] := W#16#0;
   BUFFER[55] := W#16#0;
   BUFFER[56] := W#16#0;
   BUFFER[57] := W#16#0;
   BUFFER[58] := W#16#0;
   BUFFER[59] := W#16#0;
   BUFFER[60] := W#16#0;
   BUFFER[61] := W#16#0;
   BUFFER[62] := W#16#0;
   BUFFER[63] := W#16#0;
   BUFFER[64] := W#16#0;
   BUFFER[65] := W#16#0;
   BUFFER[66] := W#16#0;
   BUFFER[67] := W#16#0;
   BUFFER[68] := W#16#0;
   BUFFER[69] := W#16#0;
   BUFFER[70] := W#16#0;
   BUFFER[71] := W#16#0;
   BUFFER[72] := W#16#0;
   BUFFER[73] := W#16#0;
   BUFFER[74] := W#16#0;
   BUFFER[75] := W#16#0;
   BUFFER[76] := W#16#0;
   BUFFER[77] := W#16#0;
   BUFFER[78] := W#16#0;
   BUFFER[79] := W#16#0;
   BUFFER[80] := W#16#0;
   BUFFER[81] := W#16#0;
   BUFFER[82] := W#16#0;
   BUFFER[83] := W#16#0;
   BUFFER[84] := W#16#0;
   BUFFER[85] := W#16#0;
   BUFFER[86] := W#16#0;
   BUFFER[87] := W#16#0;
   BUFFER[88] := W#16#0;
   BUFFER[89] := W#16#0;
   BUFFER[90] := W#16#0;
   BUFFER[91] := W#16#0;
   BUFFER[92] := W#16#0;
   BUFFER[93] := W#16#0;
   BUFFER[94] := W#16#0;
   BUFFER[95] := W#16#0;
   BUFFER[96] := W#16#0;
   BUFFER[97] := W#16#0;
   BUFFER[98] := W#16#0;
   BUFFER[99] := W#16#0;
   BUFFER[100] := W#16#0;
   BUFFER[101] := W#16#0;
   BUFFER[102] := W#16#0;
   BUFFER[103] := W#16#0;
   BUFFER[104] := W#16#0;
   BUFFER[105] := W#16#0;
   BUFFER[106] := W#16#0;
   BUFFER[107] := W#16#0;
   BUFFER[108] := W#16#0;
   BUFFER[109] := W#16#0;
   BUFFER[110] := W#16#0;
   BUFFER[111] := W#16#0;
   BUFFER[112] := W#16#0;
   BUFFER[113] := W#16#0;
   BUFFER[114] := W#16#0;
   BUFFER[115] := W#16#0;
   BUFFER[116] := W#16#0;
   BUFFER[117] := W#16#0;
   BUFFER[118] := W#16#0;
   BUFFER[119] := W#16#0;
   REASON_FOR_CLOSE := B#16#0;
   DS_NR := B#16#0;
   MAX_PUFF_LEN_SAVE := W#16#0;
   TYP_BOOL := FALSE;
   KANAL_PROBLEM := FALSE;
   KOMM_PROBLEM := FALSE;
   RECV_STARTED := FALSE;
   SEND_STARTED := FALSE;
   RESET_REQUEST := FALSE;
   RESET_EXECUTED := FALSE;
   DS200_BUSY := FALSE;
   LADDR_PTR := DW#16#0;
   LADDR := W#16#0;
   ZIEL_BYTE_SAVE := B#16#0;
   BOOL_ZIEL_BAD := FALSE;
   PARAM_OFFSET := DW#16#0;
   SLEEP := B#16#0;
   SLEEP_EXT := B#16#0;
   ID_CLOSE := W#16#0;
   RUNNING_LEN := W#16#0;
   FB_KENNUNG := B#16#F2;
END_DATA_BLOCK

ORGANIZATION_BLOCK OB 1
TITLE = "Main Program Sweep (Cycle)"
VERSION : 0.1


VAR_TEMP
  OB1_EV_CLASS : BYTE ;	//Bits 0-3 = 1 (Coming event), Bits 4-7 = 1 (Event class 1)
  OB1_SCAN_1 : BYTE ;	//1 (Cold restart scan 1 of OB 1), 3 (Scan 2-n of OB 1)
  OB1_PRIORITY : BYTE ;	//Priority of OB Execution
  OB1_OB_NUMBR : BYTE ;	//1 (Organization block 1, OB1)
  OB1_RESERVED_1 : BYTE ;	//Reserved for system
  OB1_RESERVED_2 : BYTE ;	//Reserved for system
  OB1_PREV_CYCLE : INT ;	//Cycle time of previous OB1 scan (milliseconds)
  OB1_MIN_CYCLE : INT ;	//Minimum cycle time of OB1 (milliseconds)
  OB1_MAX_CYCLE : INT ;	//Maximum cycle time of OB1 (milliseconds)
  OB1_DATE_TIME : DATE_AND_TIME ;	//Date and time OB1 started
END_VAR
BEGIN
NETWORK
TITLE =VKE0 for interruptions (only for commissioning or debugging)

      AN    OV;
      R     M      3.0;
      S     M      3.1;
      R     M      3.2;
      S     M      3.3;
NETWORK
TITLE =

      UC    FC    98;
NETWORK
TITLE =

      UC    FC   114;
NETWORK
TITLE =

      UC    FC   130;
NETWORK
TITLE =

      UC    FC   200;
NETWORK
TITLE =

      UC    FC   210;
NETWORK
TITLE =

      CALL FC   324 ;
      NOP   0;
END_ORGANIZATION_BLOCK

ORGANIZATION_BLOCK OB 82
TITLE = "I/O Point Fault"
VERSION : 0.1


VAR_TEMP
  OB82_EV_CLASS : BYTE ;	//16#39, Event class 3, Entering event state, Internal fault event
  OB82_FLT_ID : BYTE ;	//16#XX, Fault identifcation code
  OB82_PRIORITY : BYTE ;	//Priority of OB Execution
  OB82_OB_NUMBR : BYTE ;	//82 (Organization block 82, OB82)
  OB82_RESERVED_1 : BYTE ;	//Reserved for system
  OB82_IO_FLAG : BYTE ;	//Input (01010100), Output (01010101)
  OB82_MDL_ADDR : INT ;	//Base address of module with fault
  OB82_MDL_DEFECT : BOOL ;	//Module defective
  OB82_INT_FAULT : BOOL ;	//Internal fault
  OB82_EXT_FAULT : BOOL ;	//External fault
  OB82_PNT_INFO : BOOL ;	//Point information
  OB82_EXT_VOLTAGE : BOOL ;	//External voltage low
  OB82_FLD_CONNCTR : BOOL ;	//Field wiring connector missing
  OB82_NO_CONFIG : BOOL ;	//Module has no configuration data
  OB82_CONFIG_ERR : BOOL ;	//Module has configuration error
  OB82_MDL_TYPE : BYTE ;	//Type of module
  OB82_SUB_NDL_ERR : BOOL ;	//Sub-Module is missing or has error
  OB82_COMM_FAULT : BOOL ;	//Communication fault
  OB82_MDL_STOP : BOOL ;	//Module is stopped
  OB82_WTCH_DOG_FLT : BOOL ;	//Watch dog timer stopped module
  OB82_INT_PS_FLT : BOOL ;	//Internal power supply fault
  OB82_PRIM_BATT_FLT : BOOL ;	//Primary battery is in fault
  OB82_BCKUP_BATT_FLT : BOOL ;	//Backup battery is in fault
  OB82_RESERVED_2 : BOOL ;	//Reserved for system
  OB82_RACK_FLT : BOOL ;	//Rack fault, only for bus interface module
  OB82_PROC_FLT : BOOL ;	//Processor fault
  OB82_EPROM_FLT : BOOL ;	//EPROM fault
  OB82_RAM_FLT : BOOL ;	//RAM fault
  OB82_ADU_FLT : BOOL ;	//ADU fault
  OB82_FUSE_FLT : BOOL ;	//Fuse fault
  OB82_HW_INTR_FLT : BOOL ;	//Hardware interupt input in fault
  OB82_RESERVED_3 : BOOL ;	//Reserved for system
  OB82_DATE_TIME : DATE_AND_TIME ;	//Date and time OB82 started
END_VAR
BEGIN
NETWORK
TITLE =



END_ORGANIZATION_BLOCK

ORGANIZATION_BLOCK OB 85
TITLE = "Organization Block (OB) Not Loaded Fault"
VERSION : 0.1


VAR_TEMP
  OB85_EV_CLASS : BYTE ;	//16#35 Event class 3
  OB85_FLT_ID : BYTE ;	//16#XX, Fault identification code
  OB85_PRIORITY : BYTE ;	//Priority of OB Execution
  OB85_OB_NUMBR : BYTE ;	//85 (Organization block 85, OB85)
  OB85_RESERVED_1 : BYTE ;	//Reserved for system
  OB85_RESERVED_2 : BYTE ;	//Reserved for system
  OB85_RESERVED_3 : INT ;	//Reserved for system
  OB85_ERR_EV_CLASS : BYTE ;	//Class of event causing error
  OB85_ERR_EV_NUM : BYTE ;	//Number of event causing error
  OB85_OB_PRIOR : BYTE ;	//Priority of OB causing error
  OB85_OB_NUM : BYTE ;	//Number of OB causing error
  OB85_DATE_TIME : DATE_AND_TIME ;	//Date and time OB85 started
END_VAR
BEGIN
NETWORK
TITLE =



END_ORGANIZATION_BLOCK

ORGANIZATION_BLOCK OB 86
TITLE = "Loss Of Rack Fault"
VERSION : 0.1


VAR_TEMP
  OB86_EV_CLASS : BYTE ;	//16#38/39 Event class 3
  OB86_FLT_ID : BYTE ;	//16#C1/C4/C5, Fault identifcation code
  OB86_PRIORITY : BYTE ;	//Priority of OB Execution
  OB86_OB_NUMBR : BYTE ;	//86 (Organization block 86, OB86)
  OB86_RESERVED_1 : BYTE ;	//Reserved for system
  OB86_RESERVED_2 : BYTE ;	//Reserved for system
  OB86_MDL_ADDR : INT ;	//Base address of IM module in rack with fault
  OB86_RACKS_FLTD : ARRAY  [0 .. 31 ] OF BOOL ;	//Racks in fault
  OB86_DATE_TIME : DATE_AND_TIME ;	//Date and time OB86 started
END_VAR
BEGIN
NETWORK
TITLE =



END_ORGANIZATION_BLOCK

ORGANIZATION_BLOCK OB 87
TITLE = "Communication Fault"
VERSION : 0.1


VAR_TEMP
  OB87_EV_CLASS : BYTE ;	//16#39 Event class 3
  OB87_FLT_ID : BYTE ;	//16#XX, Fault identifcation code
  OB87_PRIORITY : BYTE ;	//Priority of OB Execution
  OB87_OB_NUMBR : BYTE ;	//87 (Organization block 87, OB87)
  OB87_RESERVED_1 : BYTE ;	//Reserved for system
  OB87_RESERVED_2 : BYTE ;	//Reserved for system
  OB87_RESERVED_3 : WORD ;	//Reserved for system
  OB87_RESERVED_4 : DWORD ;	//Reserved for system
  OB87_DATE_TIME : DATE_AND_TIME ;	//Date and time OB87 started
END_VAR
BEGIN
NETWORK
TITLE =



END_ORGANIZATION_BLOCK

ORGANIZATION_BLOCK OB 100
TITLE = "Complete Restart"
VERSION : 0.1


VAR_TEMP
  OB100_EV_CLASS : BYTE ;	//16#13, Event class 1, Entering event state, Event logged in diagnostic buffer
  OB100_STRTUP : BYTE ;	//16#81/82/83/84 Method of startup
  OB100_PRIORITY : BYTE ;	//Priority of OB Execution
  OB100_OB_NUMBR : BYTE ;	//100 (Organization block 100, OB100)
  OB100_RESERVED_1 : BYTE ;	//Reserved for system
  OB100_RESERVED_2 : BYTE ;	//Reserved for system
  OB100_STOP : WORD ;	//Event that caused CPU to stop (16#4xxx)
  OB100_STRT_INFO : DWORD ;	//Information on how system started
  OB100_DATE_TIME : DATE_AND_TIME ;	//Date and time OB100 started
END_VAR
BEGIN
NETWORK
TITLE =



END_ORGANIZATION_BLOCK

ORGANIZATION_BLOCK OB 121
TITLE = "Programming Error"
VERSION : 0.1


VAR_TEMP
  OB121_EV_CLASS : BYTE ;	//16#25, Event class 2, Entering event state, Internal fault event
  OB121_SW_FLT : BYTE ;	//16#XX Software programming fault
  OB121_PRIORITY : BYTE ;	//Priority of OB Execution
  OB121_OB_NUMBR : BYTE ;	//121 (Organization block 121, OB121)
  OB121_BLK_TYPE : BYTE ;	//16#88/8A/8B/8C/8E Type of block fault occured in
  OB121_RESERVED_1 : BYTE ;	//Reserved for system
  OB121_FLT_REG : WORD ;	//16#XX Specific register that caused fault
  OB121_BLK_NUM : WORD ;	//Number of block that programming fault occured in
  OB121_PRG_ADDR : WORD ;	//Address in block where programming fault occured
  OB121_DATE_TIME : DATE_AND_TIME ;	//Date and time OB121 started
END_VAR
BEGIN
NETWORK
TITLE =

END_ORGANIZATION_BLOCK

ORGANIZATION_BLOCK OB 122
TITLE = "Module Access Error"
VERSION : 0.1


VAR_TEMP
  OB122_EV_CLASS : BYTE ;	//16#29, Event class 2, Entering event state, Internal fault event
  OB122_SW_FLT : BYTE ;	//16#XX Software error code
  OB122_PRIORITY : BYTE ;	//Priority of OB Execution
  OB122_OB_NUMBR : BYTE ;	//122 (Organization block 122, OB122)
  OB122_BLK_TYPE : BYTE ;	//16#88/8C/8E Type of block fault occured in
  OB122_MEM_AREA : BYTE ;	//Memory area where access error occured
  OB122_MEM_ADDR : WORD ;	//Memory address where access error occured
  OB122_BLK_NUM : WORD ;	//Block number in which error occured
  OB122_PRG_ADDR : WORD ;	//Program address where error occured
  OB122_DATE_TIME : DATE_AND_TIME ;	//Date and time OB1 started
END_VAR
BEGIN
NETWORK
TITLE =

END_ORGANIZATION_BLOCK

